DATA_BLOCK "DB %%TAG%%"
{ S7_Optimized_Access := 'FALSE' }
VERSION : 0.1
NON_RETAIN
"@pc FB600 PID"

BEGIN
   SAMPLE_T := 0.1;
   RESTART := FALSE;
   "___ M o d e" := FALSE;
   "A/M_MODE_LINK" := FALSE;
   MODE_AUTO_LINK := FALSE;
   ENOP_SEL_MODE_MAN := TRUE;
   ENOP_SEL_MODE_AUTO := TRUE;
   ENOP_LMN_WR := TRUE;
   ENOP_SP_OP := TRUE;
   ENOP_TOSEL_INT_SP := TRUE;
   ENOP_TOSEL_EXT_SP := TRUE;
   "___ S e t p o i n t" := FALSE;
   SPINT_UPLIM := 100.0;
   SPINT_LOLIM := 0.0;
   SPEXT_UPLIM := 100.0;
   SPEXT_LOLIM := 0.0;
   LINK_SEL_SP_MODE := FALSE;
   LINK_SPEXT_MODE := FALSE;
   SETPOINT_EXT := 0.0;
   EN_TRK_SPINT_EXT := TRUE;
   EN_TRK_SPINT_PV := FALSE;
   SP_RAMP_POS := 100.0;
   SP_RAMP_NEG := 100.0;
   SP_RAMP_OFF := TRUE;
   "___ M a n i p u l a t e d  V a r" := FALSE;
   LMN_TRK := FALSE;
   LMN_TRK_SET := 0.0;
   LMN_OFFSET := 0.0;
   LMN_NM_UPLIM := 100.0;
   LMN_NM_LOLIM := 0.0;
   LMN_AUT_UPLIM := 100.0;
   LMN_AUT_LOLIM := 0.0;
   LMN_MAN_UPLIM := 100.0;
   LMN_MAN_LOLIM := 0.0;
   "___ C o n t r o l l e d  V a r" := FALSE;
   PV_UPLIM := 400.0;
   PV_LOLIM := -200.0;
   PV_IN := 20.0;
   PV_DDB := 0.0;
   DISV := 0.0;
   "___ T u n i n g  P I D" := FALSE;
   PID_GAIN_EN := TRUE;
   PID_GAIN := 0.8;
   PID_GAIN_REV := FALSE;
   PID_GAIN_PFDB_SEL := FALSE;
   PID_TI := 10.0;
   PID_INT_HPOS := FALSE;
   PID_INT_HNEG := FALSE;
   PID_TD := 0.0;
   PID_D_PFDB_SEL := FALSE;
   PID_TIME_LAG := 1.0;
   "___ A l a r m" := FALSE;
   EN_ALM_PVUP := TRUE;
   EN_ALM_PVLO := TRUE;
   SET_ALM_PVUP := 100.0;
   SET_ALM_PVLO := -100.0;
   ALM_HYS := 0.1;
   SET_DLY_ALM_PVUP := 0.0;
   SET_DLY_ALM_PVLO := 0.0;
   Q_SPRAMP_POSLIM_ON := FALSE;
   Q_SPRAMP_NEGLIM_ON := FALSE;
   Q_SP_HLIMIT_ON := FALSE;
   Q_SP_LLIMIT_ON := FALSE;
   Q_OP_ENABLED_SP := TRUE;
   Q_SP_IS_EXT := FALSE;
   Q_OP_ENABLED_SEL_INT := TRUE;
   Q_OP_ENABLED_SEL_EXT := TRUE;
   Q_LMN_UPLIM_ON := FALSE;
   Q_LMN_LOLIM_ON := TRUE;
   Q_OP_ENABLED_LMN := FALSE;
   Q_AUTO_MODE_ON := TRUE;
   Q_OP_ENABLED_MANMODE := TRUE;
   Q_OP_ENABLED_AUTOMODE := TRUE;
   Q_CAS_CUT := TRUE;
   Q_ERR_ALM_PVUP := FALSE;
   Q_HMI_ALM_PVUP := FALSE;
   Q_ERR_ALM_PVLO := FALSE;
   Q_HMI_ALM_PVLO := FALSE;
   Q_LMN := 0.0;
   Q_ER := 10.0;
   Q_SP := 30.0;
   W_ALM := 16#0000;
   LMM_MAN_OPSET := 0.0;
   SETPOINT_INT := 30.0;
   HMISEL_EXT := FALSE;
   HMISEL_AUTO_MODE := TRUE;
   sbOPD1_I0 := FALSE;
   sbOPD2_I0 := TRUE;
   sbQERH_ALM := FALSE;
   sbQERL_ALM := FALSE;
   sbQLMN_HLM := FALSE;
   sbQLMN_LLM := TRUE;
   sInvAlt := -1.333333;
   sIanteilAlt := 1.321667;
   sRestInt := 0.0;
   sRestDif := 0.0;
   sRueck := -1.333333;
   sSpOld := 30.0;
   OP_A_SP.OP_EN := TRUE;
   OP_A_SP.U_HL := 100.0;
   OP_A_SP.U_LL := 0.0;
   OP_A_SP.LINK_U := 30.0;
   OP_A_SP.LINK_ON := FALSE;
   OP_A_SP.BTRACK := TRUE;
   OP_A_SP.V := 30.0;
   OP_A_SP.QOP_EN := TRUE;
   OP_A_SP.QVHL := FALSE;
   OP_A_SP.QVLL := FALSE;
   OP_A_SP.U := 30.0;
   OP_A_SP.srU := 30.0;
   OP_A_SP.sbRESTART := FALSE;
   OP_A_MAN.OP_EN := TRUE;
   OP_A_MAN.U_HL := 100.0;
   OP_A_MAN.U_LL := 0.0;
   OP_A_MAN.LINK_U := 0.0;
   OP_A_MAN.LINK_ON := TRUE;
   OP_A_MAN.BTRACK := TRUE;
   OP_A_MAN.V := 0.0;
   OP_A_MAN.QOP_EN := FALSE;
   OP_A_MAN.QVHL := FALSE;
   OP_A_MAN.QVLL := FALSE;
   OP_A_MAN.U := 0.0;
   OP_A_MAN.srU := 0.0;
   OP_A_MAN.sbRESTART := FALSE;
   dwDUMMY := 16#0000_0000;
   QERL_ALM_TIMER_P.SAMPLE_T := 0.1;
   QERL_ALM_TIMER_P.TIME0 := 0.0;
   QERL_ALM_TIMER_P.MODE := 2;
   QERL_ALM_TIMER_P.RESET := FALSE;
   QERL_ALM_TIMER_P.I0 := FALSE;
   QERL_ALM_TIMER_P.QERR := FALSE;
   QERL_ALM_TIMER_P.Q0 := FALSE;
   QERL_ALM_TIMER_P.PTIME := 0.0;
   QERL_ALM_TIMER_P.ETIME := 0.0;
   QERL_ALM_TIMER_P.ACTIVE := FALSE;
   QERL_ALM_TIMER_P.I0_FP := FALSE;
   QERL_ALM_TIMER_P.I0_MODE1_FP := FALSE;
   QERL_ALM_TIMER_P.I0_MODE3_FP := FALSE;
   QERH_ALM_TIMER_P.SAMPLE_T := 0.1;
   QERH_ALM_TIMER_P.TIME0 := 0.0;
   QERH_ALM_TIMER_P.MODE := 2;
   QERH_ALM_TIMER_P.RESET := FALSE;
   QERH_ALM_TIMER_P.I0 := FALSE;
   QERH_ALM_TIMER_P.QERR := FALSE;
   QERH_ALM_TIMER_P.Q0 := FALSE;
   QERH_ALM_TIMER_P.PTIME := 0.0;
   QERH_ALM_TIMER_P.ETIME := 0.0;
   QERH_ALM_TIMER_P.ACTIVE := FALSE;
   QERH_ALM_TIMER_P.I0_FP := FALSE;
   QERH_ALM_TIMER_P.I0_MODE1_FP := FALSE;
   QERH_ALM_TIMER_P.I0_MODE3_FP := FALSE;
   TAG := '%%TAG%%';
   DESCR := '%%DESC%%';
   UM_PV := '%%UNIT%%';
   UM_LMN := '%';

END_DATA_BLOCK

